_CFC_ (* Continuous Function Chart, elements in execution order *)
#0 RT_Auto:R_TRIG(CLK: SCHU_P2_2_UST_AUTO_VH)
#1 RT_Zima:R_TRIG(CLK: SCHU_P2_2_UST_LETO_VH)
#2 RT_Leto:R_TRIG(CLK: SCHU_P2_2_UST_ZIMA_VH)
#3 OR(#1.Q, #2.Q)
#4 RS_Auto:RS(SET: #12, RESET1: #3)
#5 AND(SCHU_P2_2_TE1_B_UST_SEZ_LETO, #4.Q1)
#6 OR(#1.Q, #5)
#7 AND(#4.Q1, SCHU_P2_2_TE1_M_UST_SEZ_LETO)
#8 OR(#7, #2.Q)
#9 RS_Sezon:RS(SET: #6, RESET1: #8)
#10 SCHU_P2_2_UST_LETO <= #9.Q1
#11 SCHU_P2_2_UST_ZIMA <= NOT #9.Q1
#12 OR(#15.Q, #0.Q)
#13 SCHU_P2_2_UST_SOST_AUTO <= #4.Q1
#14 SCHU_P2_2_UST_SOST_DIST <= NOT #4.Q1
#15 RT_T:R_TRIG(CLK: TRUE)
_END_CFC_
(* the same logic as Structured Text *)
RT_Auto(CLK := SCHU_P2_2_UST_AUTO_VH);
RT_Zima(CLK := SCHU_P2_2_UST_LETO_VH);
RT_Leto(CLK := SCHU_P2_2_UST_ZIMA_VH);
RS_Auto(SET := _t72, RESET1 := RT_Zima.Q OR RT_Leto.Q);
RS_Sezon(SET := RT_Zima.Q OR (SCHU_P2_2_TE1_B_UST_SEZ_LETO AND RS_Auto.Q1), RESET1 := (RS_Auto.Q1 AND SCHU_P2_2_TE1_M_UST_SEZ_LETO) OR RT_Leto.Q);
SCHU_P2_2_UST_LETO := RS_Sezon.Q1;
SCHU_P2_2_UST_ZIMA := NOT RS_Sezon.Q1;
_t72 := RT_T.Q OR RT_Auto.Q;
SCHU_P2_2_UST_SOST_AUTO := RS_Auto.Q1;
SCHU_P2_2_UST_SOST_DIST := NOT RS_Auto.Q1;
RT_T(CLK := TRUE);
END_PROGRAM

(* POU Regim/Sost, CFC *)
PROGRAM Sost
VAR
	RS_Sost: RS;
	RT_PUSK: R_TRIG;
	RT_STOP: R_TRIG;
	RS_Old_Sost: RS;
	TON_Kv1: TON;
	TON_Kv1_1: TON;
	OLD_SOST: BOOL;

	KV1: BOOL;
	RT_PUSK_OLD: R_TRIG;
	CTU_TS: CTU;
	TOF_TS_1: TOF;
	TOF_TS_2: TOF;
	TOF_TS_3: TOF;
	RT_PUSK_OLD1: R_TRIG;
	TON_Kv1_11: TON;
	TON_Kv11: TON;
	TOF_TE_1: TOF;
	TOF_Te_2: TOF;
	TOF_Te_3: TOF;
	CTU_Te: CTU;
END_VAR
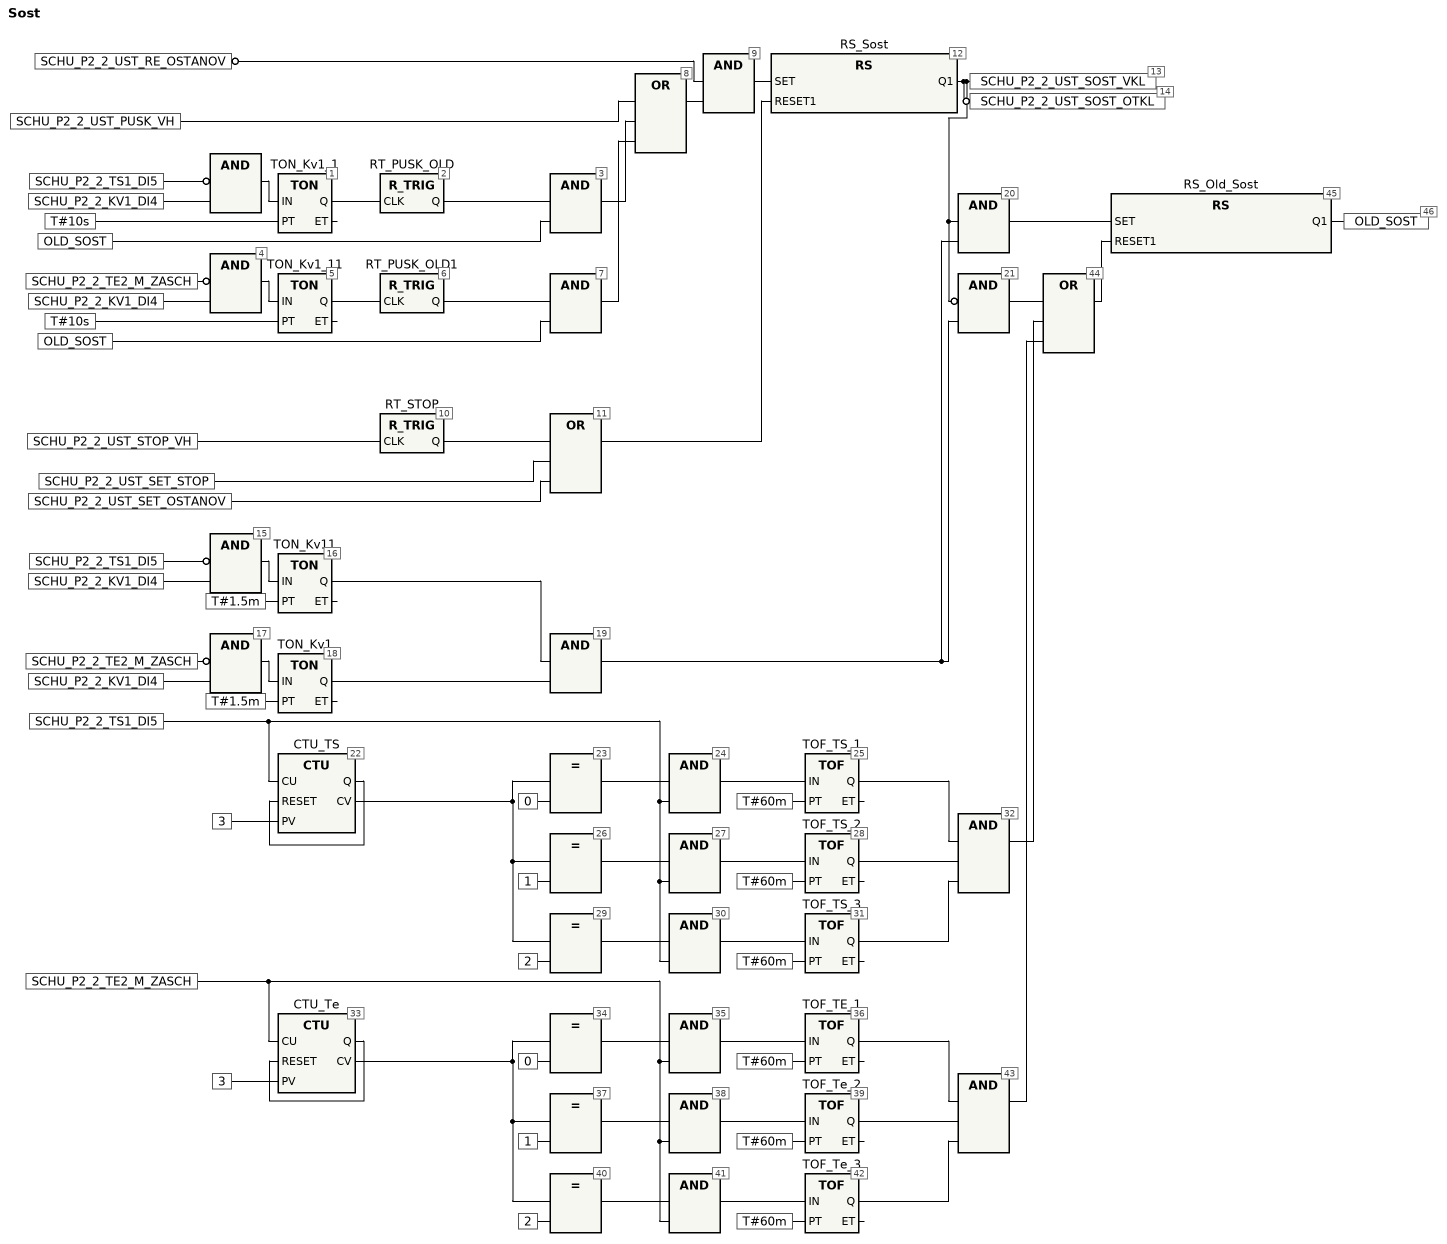
